// TIA Portal V20 export
FUNCTION_BLOCK "Main_Safety_RTG1"   // FB30, F_LAD
{ S7_Optimized_Access := 'TRUE' }
// ============================================================================
// // POSALUX Swiss SA / (C) Copyright 2024
// //----------------------------------------------------------------------------------
// // Title: Programme Principale Safety
// // Comment/Function: 
// //
// // Author: Olivier Heim
// // Engineering: TIA Portal v17
// //----------------------------------------------------------------------------------
// // Change log table:
// // Version   | Date            | Expert in charge | Changes applied
// // -----------------|---------------------|--------------------------------|------------------------------------
// // 00.00.01 | 20241218 | HOL                        | First released version
// // -----------------|---------------------|--------------------------------|------------------------------------
// // 01.01.00 | 20241218 | FMI                         | General improves
// / ============================================================================
// stored: AutoNumber false
   VAR
      sSupplyPower : Bool;
      sAckEmergencyStop : Bool;
      sAckFdbPowMach : Bool;
      sAckFdbBW_LoaderEstopRelay : Bool;
      sAckFdbSonplasDoorClosedRelay : Bool;
      ESTOP1_Instance : ESTOP1;
      FDBACK_PowerMachine : FDBACK;
      FDBACK_BW_LoaderEstopRelay : FDBACK;
      FDBACK_SonplasDoorClosedRelay : FDBACK;
      DB_ACK_GL : ACK_GL;
   END_VAR
BEGIN

REGION Network 1: Transfer DataToSafety to DataToSafety F
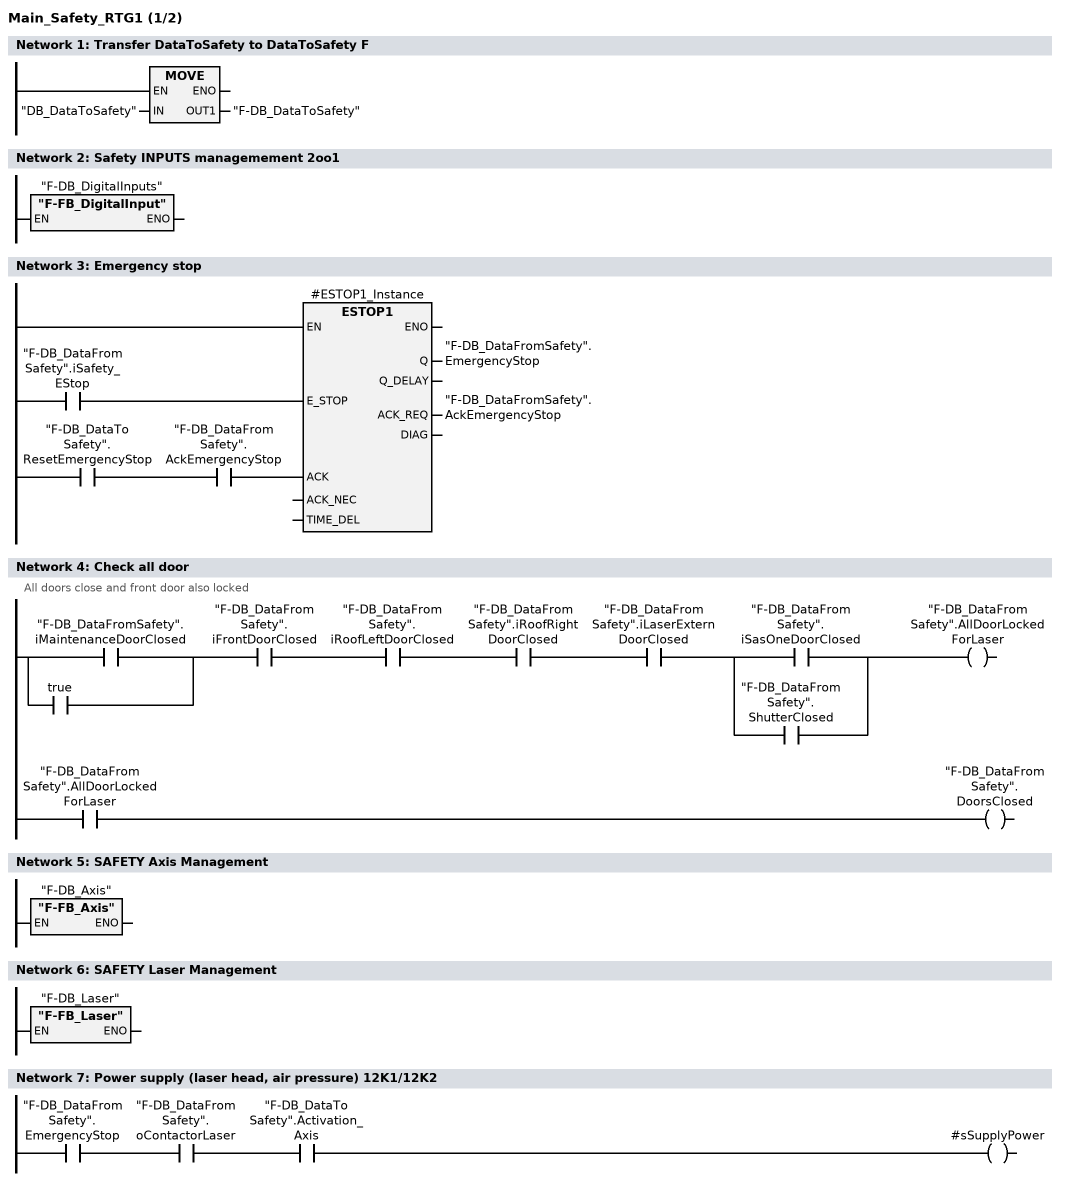
   RUNG wire#powerrail
      { S7_GenerateENO := "TRUE" } Move(in := "DB_DataToSafety", out1 => "F-DB_DataToSafety")
   END_RUNG
   // the same network as SCL:
   "F-DB_DataToSafety" := "DB_DataToSafety";
END_REGION

REGION Network 2: Safety INPUTS managemement 2oo1
   RUNG wire#powerrail
      "F-DB_DigitalInputs"()
   END_RUNG
   // the same network as SCL:
   "F-DB_DigitalInputs"();   // "F-FB_DigitalInput"
END_REGION

REGION Network 3: Emergency stop
   RUNG wire#powerrail
      #ESTOP1_Instance.ESTOP1(E_STOP := wire#w1, ACK := wire#w2, ACK_NEC :=, TIME_DEL :=, Q => "F-DB_DataFromSafety".EmergencyStop, Q_DELAY =>, ACK_REQ => "F-DB_DataFromSafety".AckEmergencyStop, DIAG =>)
   END_RUNG
   RUNG wire#powerrail
      Contact( "F-DB_DataFromSafety".iSafety_EStop )
   END_RUNG wire#w1
   RUNG wire#powerrail
      Contact( "F-DB_DataToSafety".ResetEmergencyStop )
      Contact( "F-DB_DataFromSafety".AckEmergencyStop )
   END_RUNG wire#w2
   // the same network as SCL:
   #ESTOP1_Instance(E_STOP := "F-DB_DataFromSafety".iSafety_EStop,   // ESTOP1
                    ACK := "F-DB_DataToSafety".ResetEmergencyStop AND "F-DB_DataFromSafety".AckEmergencyStop,
                    Q => "F-DB_DataFromSafety".EmergencyStop,
                    ACK_REQ => "F-DB_DataFromSafety".AckEmergencyStop);
END_REGION

REGION Network 4: Check all door
   // All doors close and front door also locked
   RUNG wire#powerrail
      Contact( "F-DB_DataFromSafety".iMaintenanceDoorClosed )
      wire#w1
      Contact( "F-DB_DataFromSafety".iFrontDoorClosed )
      Contact( "F-DB_DataFromSafety".iRoofLeftDoorClosed )
      Contact( "F-DB_DataFromSafety".iRoofRightDoorClosed )
      Contact( "F-DB_DataFromSafety".iLaserExternDoorClosed )
      wire#w2
      Contact( "F-DB_DataFromSafety".iSasOneDoorClosed )
      wire#w3
      Coil( "F-DB_DataFromSafety".AllDoorLockedForLaser )
   END_RUNG
   RUNG wire#powerrail
      Contact( true )
   END_RUNG wire#w1
   RUNG wire#w2
      Contact( "F-DB_DataFromSafety".ShutterClosed )
   END_RUNG wire#w3
   RUNG wire#powerrail
      Contact( "F-DB_DataFromSafety".AllDoorLockedForLaser )
      Coil( "F-DB_DataFromSafety".DoorsClosed )
   END_RUNG
   // the same network as SCL:
   "F-DB_DataFromSafety".AllDoorLockedForLaser := ("F-DB_DataFromSafety".iMaintenanceDoorClosed OR true) AND "F-DB_DataFromSafety".iFrontDoorClosed AND "F-DB_DataFromSafety".iRoofLeftDoorClosed AND "F-DB_DataFromSafety".iRoofRightDoorClosed AND "F-DB_DataFromSafety".iLaserExternDoorClosed AND ("F-DB_DataFromSafety".iSasOneDoorClosed OR "F-DB_DataFromSafety".ShutterClosed);
   "F-DB_DataFromSafety".DoorsClosed := "F-DB_DataFromSafety".AllDoorLockedForLaser;
END_REGION

REGION Network 5: SAFETY Axis Management
   RUNG wire#powerrail
      "F-DB_Axis"()
   END_RUNG
   // the same network as SCL:
   "F-DB_Axis"();   // "F-FB_Axis"
END_REGION

REGION Network 6: SAFETY Laser Management
   RUNG wire#powerrail
      "F-DB_Laser"()
   END_RUNG
   // the same network as SCL:
   "F-DB_Laser"();   // "F-FB_Laser"
END_REGION

REGION Network 7: Power supply (laser head, air pressure) 12K1/12K2
   RUNG wire#powerrail
      Contact( "F-DB_DataFromSafety".EmergencyStop )
      Contact( "F-DB_DataFromSafety".oContactorLaser )
      Contact( "F-DB_DataToSafety".Activation_Axis )
      Coil( #sSupplyPower )
   END_RUNG
   // the same network as SCL:
   #sSupplyPower := "F-DB_DataFromSafety".EmergencyStop AND "F-DB_DataFromSafety".oContactorLaser AND "F-DB_DataToSafety".Activation_Axis;
END_REGION

REGION Network 8: Check feed back power supply
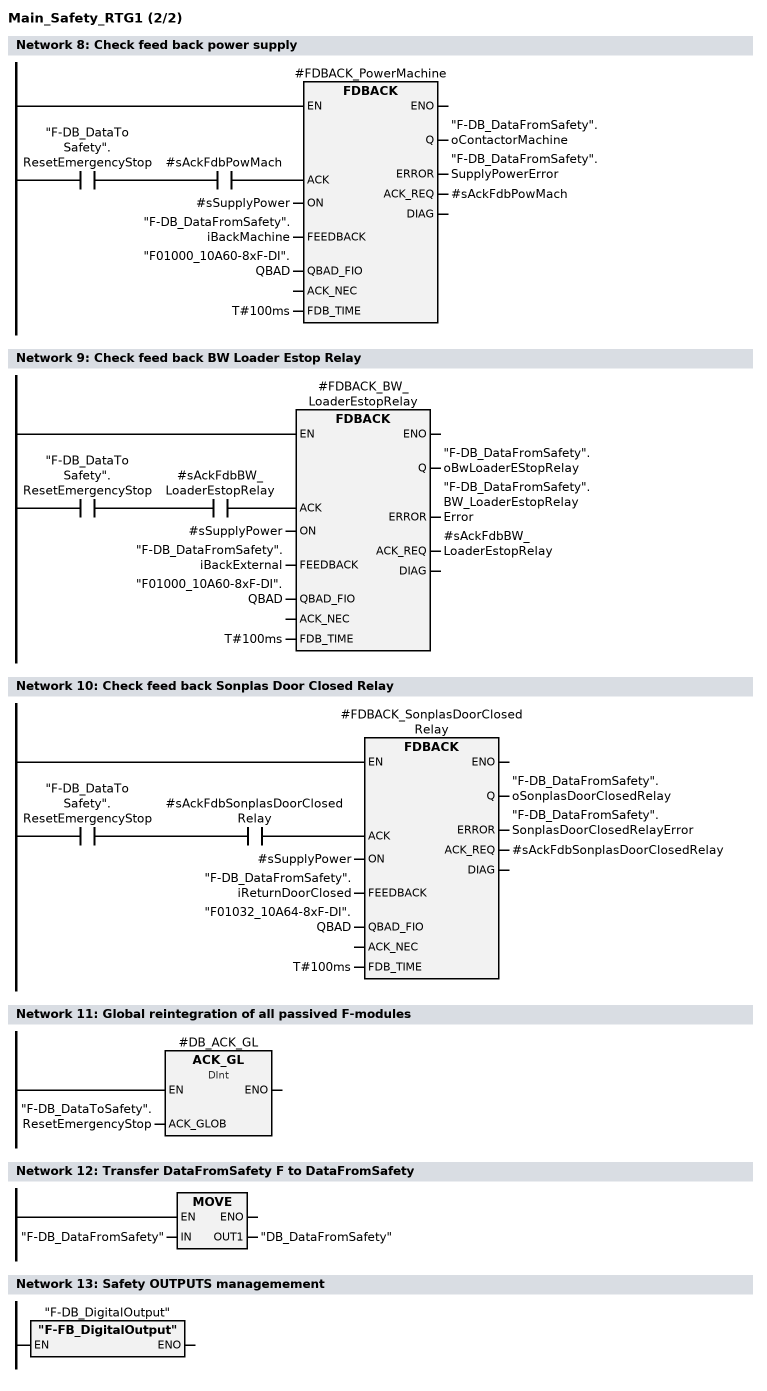
   RUNG wire#powerrail
      #FDBACK_PowerMachine.FDBACK(ACK := wire#w1, ON := #sSupplyPower, FEEDBACK := "F-DB_DataFromSafety".iBackMachine, QBAD_FIO := "F01000_10A60-8xF-DI".QBAD, ACK_NEC :=, FDB_TIME := T#100ms, Q => "F-DB_DataFromSafety".oContactorMachine, ERROR => "F-DB_DataFromSafety".SupplyPowerError, ACK_REQ => #sAckFdbPowMach, DIAG =>)
   END_RUNG
   RUNG wire#powerrail
      Contact( "F-DB_DataToSafety".ResetEmergencyStop )
      Contact( #sAckFdbPowMach )
   END_RUNG wire#w1
   // the same network as SCL:
   #FDBACK_PowerMachine(ACK := "F-DB_DataToSafety".ResetEmergencyStop AND #sAckFdbPowMach,   // FDBACK
                        ON := #sSupplyPower,
                        FEEDBACK := "F-DB_DataFromSafety".iBackMachine,
                        QBAD_FIO := "F01000_10A60-8xF-DI".QBAD,
                        FDB_TIME := T#100ms,
                        Q => "F-DB_DataFromSafety".oContactorMachine,
                        ERROR => "F-DB_DataFromSafety".SupplyPowerError,
                        ACK_REQ => #sAckFdbPowMach);
END_REGION

REGION Network 9: Check feed back BW Loader Estop Relay
   RUNG wire#powerrail
      #FDBACK_BW_LoaderEstopRelay.FDBACK(ACK := wire#w1, ON := #sSupplyPower, FEEDBACK := "F-DB_DataFromSafety".iBackExternal, QBAD_FIO := "F01000_10A60-8xF-DI".QBAD, ACK_NEC :=, FDB_TIME := T#100ms, Q => "F-DB_DataFromSafety".oBwLoaderEStopRelay, ERROR => "F-DB_DataFromSafety".BW_LoaderEstopRelayError, ACK_REQ => #sAckFdbBW_LoaderEstopRelay, DIAG =>)
   END_RUNG
   RUNG wire#powerrail
      Contact( "F-DB_DataToSafety".ResetEmergencyStop )
      Contact( #sAckFdbBW_LoaderEstopRelay )
   END_RUNG wire#w1
   // the same network as SCL:
   #FDBACK_BW_LoaderEstopRelay(ACK := "F-DB_DataToSafety".ResetEmergencyStop AND #sAckFdbBW_LoaderEstopRelay,   // FDBACK
                           ON := #sSupplyPower,
                           FEEDBACK := "F-DB_DataFromSafety".iBackExternal,
                           QBAD_FIO := "F01000_10A60-8xF-DI".QBAD,
                           FDB_TIME := T#100ms,
                           Q => "F-DB_DataFromSafety".oBwLoaderEStopRelay,
                           ERROR => "F-DB_DataFromSafety".BW_LoaderEstopRelayError,
                           ACK_REQ => #sAckFdbBW_LoaderEstopRelay);
END_REGION

REGION Network 10: Check feed back Sonplas Door Closed Relay
   RUNG wire#powerrail
      #FDBACK_SonplasDoorClosedRelay.FDBACK(ACK := wire#w1, ON := #sSupplyPower, FEEDBACK := "F-DB_DataFromSafety".iReturnDoorClosed, QBAD_FIO := "F01032_10A64-8xF-DI".QBAD, ACK_NEC :=, FDB_TIME := T#100ms, Q => "F-DB_DataFromSafety".oSonplasDoorClosedRelay, ERROR => "F-DB_DataFromSafety".SonplasDoorClosedRelayError, ACK_REQ => #sAckFdbSonplasDoorClosedRelay, DIAG =>)
   END_RUNG
   RUNG wire#powerrail
      Contact( "F-DB_DataToSafety".ResetEmergencyStop )
      Contact( #sAckFdbSonplasDoorClosedRelay )
   END_RUNG wire#w1
   // the same network as SCL:
   #FDBACK_SonplasDoorClosedRelay(ACK := "F-DB_DataToSafety".ResetEmergencyStop AND #sAckFdbSonplasDoorClosedRelay,   // FDBACK
                           ON := #sSupplyPower,
                           FEEDBACK := "F-DB_DataFromSafety".iReturnDoorClosed,
                           QBAD_FIO := "F01032_10A64-8xF-DI".QBAD,
                           FDB_TIME := T#100ms,
                           Q => "F-DB_DataFromSafety".oSonplasDoorClosedRelay,
                           ERROR => "F-DB_DataFromSafety".SonplasDoorClosedRelayError,
                           ACK_REQ => #sAckFdbSonplasDoorClosedRelay);
END_REGION

REGION Network 11: Global reintegration of all passived F-modules
   RUNG wire#powerrail
      { S7_Templates := "codedbool_type := DInt" } #DB_ACK_GL.ACK_GL(ACK_GLOB := "F-DB_DataToSafety".ResetEmergencyStop)
   END_RUNG
   // the same network as SCL:
   #DB_ACK_GL(ACK_GLOB := "F-DB_DataToSafety".ResetEmergencyStop);   // ACK_GL
END_REGION

REGION Network 12: Transfer DataFromSafety F to DataFromSafety
   RUNG wire#powerrail
      { S7_GenerateENO := "TRUE" } Move(in := "F-DB_DataFromSafety", out1 => "DB_DataFromSafety")
   END_RUNG
   // the same network as SCL:
   "DB_DataFromSafety" := "F-DB_DataFromSafety";
END_REGION

REGION Network 13: Safety OUTPUTS managemement
   RUNG wire#powerrail
      "F-DB_DigitalOutput"()
   END_RUNG
   // the same network as SCL:
   "F-DB_DigitalOutput"();   // "F-FB_DigitalOutput"
END_REGION
END_FUNCTION_BLOCK
